FUNCTION_BLOCK Stack
VAR_INPUT
END_VAR
VAR_OUTPUT
	o_slidingCylinder : MonostableCylinder;
END_VAR
VAR
	//Sensors
	m_Presencesensor : PresenceSensor;
	m_Opticalsensor : OpticalSensor;
	m_Inductivesensor : InductiveSensor;
	m_Weightsensor : WeightSensor;
END_VAR

PROPERTY LightWPOnTray : BOOL
GET
LightWPOnTray:=m_Opticalsensor.Value;
END_GET
END_PROPERTY

PROPERTY MetalWPOnTray : BOOL
GET
MetalWPOnTray := m_Inductivesensor.Value;
END_GET
END_PROPERTY

PROPERTY WPOnTray : BOOL
 //REFERENCE TO PresenceSensor
GET
WPOnTray:=m_Presencesensor.Value;
END_GET
END_PROPERTY

PROPERTY WPWeight : INT
GET
WPWeight:=m_Weightsensor.Value;
END_GET
END_PROPERTY

END_FUNCTION_BLOCK

(* stored: Version 1.1.0.1
   POU Stack: Id {1e3fa84f-9e42-4403-ad18-2b7e89b35a5e}, SpecialFunc None
   Property LightWPOnTray: Id {c68d4113-17be-4d3a-a9fd-e1465f07ef87}
   Get Get: Id {79b9e079-4f7b-402e-8feb-229e8b73d1f0}
   Property MetalWPOnTray: Id {4bf79261-dbde-4bb0-839a-4a5690f0b9bf}
   Get Get: Id {dcf5fe41-2293-481b-b2b5-ff6139360ce0}
   Property WPOnTray: Id {7075c1af-0b9e-4f28-93a5-c96b5aa3fd9a}
   Get Get: Id {6f5e7b24-0509-4eba-a08d-b26553b408f9}
   Property WPWeight: Id {dac3abdf-3167-4b0b-b57f-f9aa92356f1d}
   Get Get: Id {b5c4852c-da2b-4ac3-a10f-6ce429dd0e84} *)
